TYPE OutputBase_10CEE7DE :
STRUCT
END_STRUCT
END_TYPE

(* stored: Version 1.2.0.0, ProductVersion 3.1.4024.11
   DUT OutputBase_10CEE7DE: Id {503989df-6cda-441e-85f5-ecbdcefb1989} *)
